Staubli VAL3: delete.pgx

public program delete(string x_sName, num& x_nResult[])
  local string l_sItem
  local num l_nSize
begin
  //
  // delete the select trajectory
  //
  if isDefined(pt:tTraj[x_sName])
    // delete
    delete(pt:tTraj[x_sName])
    // save it
    bToSave=true
    x_nResult=0
  else
    x_nResult=-1
  endIf
end
